{attribute 'qualified_only'}
VAR_GLOBAL
END_VAR

(* stored: Version 1.1.0.1, ProductVersion 3.1.4024.16
   GVL Global: Id {9f62ad20-46af-4634-87f4-f0b7f87586e9} *)
